(*******************************************************************************
                          protoc-gen-twincat V0.0.0.0                           
                  https://github.com/TcHaxx/protoc-gen-twincat                  
*******************************************************************************)
{attribute 'no-analysis'}
TYPE ST_SensorReading :
STRUCT
	value : LREAL;
	precision : REAL;
	timestamp : LINT;
END_STRUCT
END_TYPE

(* stored: Version 1.1.0.1
   DUT ST_SensorReading: Id 21507ef9-2dfc-4448-84ab-65133cf39e6e *)
